// TIA Portal V17 export
// export: Created 2024-01-30T08:49:14.8899555Z, ExportSetting WithDefaults, DisplayName Totally Integrated Automation Portal, DisplayVersion V17 Update 6, DisplayName TIA Portal Openness, DisplayVersion V17 Update 6, DisplayName TIA Portal Version Control Interface, DisplayVersion V17, DisplayName STEP 7 Professional, DisplayVersion V17 Update 6, DisplayName STEP 7 Safety, DisplayVersion V17 Update 6, DisplayName WinCC Advanced, DisplayVersion V17 Update 6
FUNCTION_BLOCK "Test_SQ"   // FB8, GRAPH
VERSION : 0.1
// stored: AcknowledgeErrorsRequired true, AutoNumber true, GraphVersion 6.0, InitialValuesAcquisition false, IsIECCheckEnabled false, LanguageInNetworks FBD, LockOperatingMode false, PermanentILProcessingInMANMode false, SetENOAutomatically false, SkipSteps false, UDAEnableTagReadback false, WithAlarmHandling true
   // inherited from GRAPH_BASE
   VAR
      OFF_SQ_BASE : Bool;
   END_VAR
   VAR_INPUT
      OFF_SQ { ExternalAccessible := 'False'; ExternalVisible := 'False'; ExternalWritable := 'False'} : Bool := false;   // Kette ausschalten
      INIT_SQ { ExternalAccessible := 'False'; ExternalVisible := 'False'; ExternalWritable := 'False'} : Bool := false;   // Kette in Initialzustand versetzen
      ACK_EF { ExternalAccessible := 'False'; ExternalVisible := 'False'; ExternalWritable := 'False'} : Bool := false;   // Alle Fehler und Störungen quittieren
      S_PREV { ExternalAccessible := 'False'; ExternalVisible := 'False'; ExternalWritable := 'False'} : Bool := false;   // Vorherigen Schritt am Parameter S_NO ausgeben
      S_NEXT { ExternalAccessible := 'False'; ExternalVisible := 'False'; ExternalWritable := 'False'} : Bool := false;   // Nächsten Schritt am Parameter S_NO anzeigen
      SW_AUTO { ExternalAccessible := 'False'; ExternalVisible := 'False'; ExternalWritable := 'False'} : Bool := false;   // Automatischer Betrieb
      SW_TAP { ExternalAccessible := 'False'; ExternalVisible := 'False'; ExternalWritable := 'False'} : Bool := false;   // Halbautomatisch/Weiterschalten mit Transition
      SW_TOP { ExternalAccessible := 'False'; ExternalVisible := 'False'; ExternalWritable := 'False'} : Bool := false;   // Halbautomatisch/Ignoriere Transition
      SW_MAN { ExternalAccessible := 'False'; ExternalVisible := 'False'; ExternalWritable := 'False'} : Bool := false;   // Handbetrieb
      S_SEL { ExternalAccessible := 'False'; ExternalVisible := 'False'; ExternalWritable := 'False'} : Int := 0;   // Schritt auswählen, der an S_NO ausgegeben werden soll
      S_ON { ExternalAccessible := 'False'; ExternalVisible := 'False'; ExternalWritable := 'False'} : Bool := false;   // Schritt aktivieren, der an Parameter S_NO anliegt
      S_OFF { ExternalAccessible := 'False'; ExternalVisible := 'False'; ExternalWritable := 'False'} : Bool := false;   // Schritt deaktivieren, der an Parameter S_NO anliegt
      T_PUSH { ExternalAccessible := 'False'; ExternalVisible := 'False'; ExternalWritable := 'False'} : Bool := false;   // Schaltfreigabe für Transition im halbautomatischen Betrieb
   END_VAR
   VAR_OUTPUT
      S_NO { ExternalAccessible := 'False'; ExternalVisible := 'False'; ExternalWritable := 'False'} : Int := 0;   // Schrittnummer
      S_MORE { ExternalAccessible := 'False'; ExternalVisible := 'False'; ExternalWritable := 'False'} : Bool := false;   // Weitere Schritte sind vorhanden und können in S_NO angezeigt werden.
      S_ACTIVE { ExternalAccessible := 'False'; ExternalVisible := 'False'; ExternalWritable := 'False'} : Bool := false;   // Schritt, der an Parameter S_NO angezeigt wird, ist aktiv
      ERR_FLT { ExternalAccessible := 'False'; ExternalVisible := 'False'; ExternalWritable := 'False'} : Bool := false;   // Sammelfehler Interlock oder Supervision
      AUTO_ON { ExternalAccessible := 'False'; ExternalVisible := 'False'; ExternalWritable := 'False'} : Bool := false;   // Automatischer Betrieb eingeschaltet
      TAP_ON { ExternalAccessible := 'False'; ExternalVisible := 'False'; ExternalWritable := 'False'} : Bool := false;   // Halbautomatischer Betrieb/Schritt mit Transition eingeschaltet
      TOP_ON { ExternalAccessible := 'False'; ExternalVisible := 'False'; ExternalWritable := 'False'} : Bool := false;   // Halbautomatischer Betrieb/Ignoriere Transition eingeschaltet
      MAN_ON { ExternalAccessible := 'False'; ExternalVisible := 'False'; ExternalWritable := 'False'} : Bool := false;   // Handbetrieb eingeschaltet
   END_VAR
BEGIN
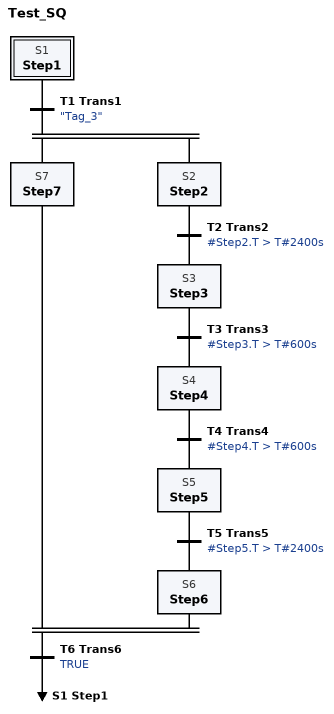
   // sequencer 1
   INITIAL_STEP Step1:   // S1, max time T#10S, warning time T#7S
   END_STEP
   TRANSITION Trans1 FROM Step1 TO (Step7, Step2)   // T1
      := "Tag_3";
   END_TRANSITION
   STEP Step2:   // S2, max time T#10S, warning time T#7S
   END_STEP
   TRANSITION Trans2 FROM Step2 TO Step3   // T2
      := #Step2.T > T#2400s;
   END_TRANSITION
   STEP Step3:   // S3, max time T#10S, warning time T#7S
   END_STEP
   TRANSITION Trans3 FROM Step3 TO Step4   // T3
      := #Step3.T > T#600s;
   END_TRANSITION
   STEP Step4:   // S4, max time T#10S, warning time T#7S
   END_STEP
   TRANSITION Trans4 FROM Step4 TO Step5   // T4
      := #Step4.T > T#600s;
   END_TRANSITION
   STEP Step5:   // S5, max time T#10S, warning time T#7S
   END_STEP
   TRANSITION Trans5 FROM Step5 TO Step6   // T5
      := #Step5.T > T#2400s;
   END_TRANSITION
   STEP Step6:   // S6, max time T#10S, warning time T#7S
   END_STEP
   STEP Step7:   // S7, max time T#10S, warning time T#7S
   END_STEP
   TRANSITION Trans6 FROM (Step6, Step7) TO Step1   // T6, jump
      := TRUE;
   END_TRANSITION
END_FUNCTION_BLOCK
